// Mitsubishi GX Works2 project: 2023-06-07 #1 생산자동화기능사 13번   PLC: Q03UDV
// 생산자동화기능사

// global labels: Global1
VAR_GLOBAL
  PB1 AT X0 : BOOL;
  PB2 AT X1 : BOOL;
  정지 AT X2 : BOOL;
  공급후진 AT X3 : BOOL;
  공급전진 AT X4 : BOOL;
  가공후진 AT X5 : BOOL;
  가공전진 AT X6 : BOOL;
  송출후진 AT X7 : BOOL;
  송출전진 AT X8 : BOOL;
  배출후진 AT X9 : BOOL;
  배출전진 AT X0A : BOOL;
  매거진 AT X0B : BOOL;
  금속센서 AT X0F : BOOL;
  PB3 AT X10 : BOOL;
  적색 AT Y20 : BOOL;
  황색 AT Y21 : BOOL;
  녹색 AT Y22 : BOOL;
  공급1 AT Y23 : BOOL;
  공급2 AT Y24 : BOOL;
  가공 AT Y25 : BOOL;
  드릴 AT Y26 : BOOL;
  송출 AT Y27 : BOOL;
  배출 AT Y28 : BOOL;
  컨베이어 AT Y29 : BOOL;
END_VAR

PROGRAM 테스트동작
VAR
  prog : INT;
END_VAR
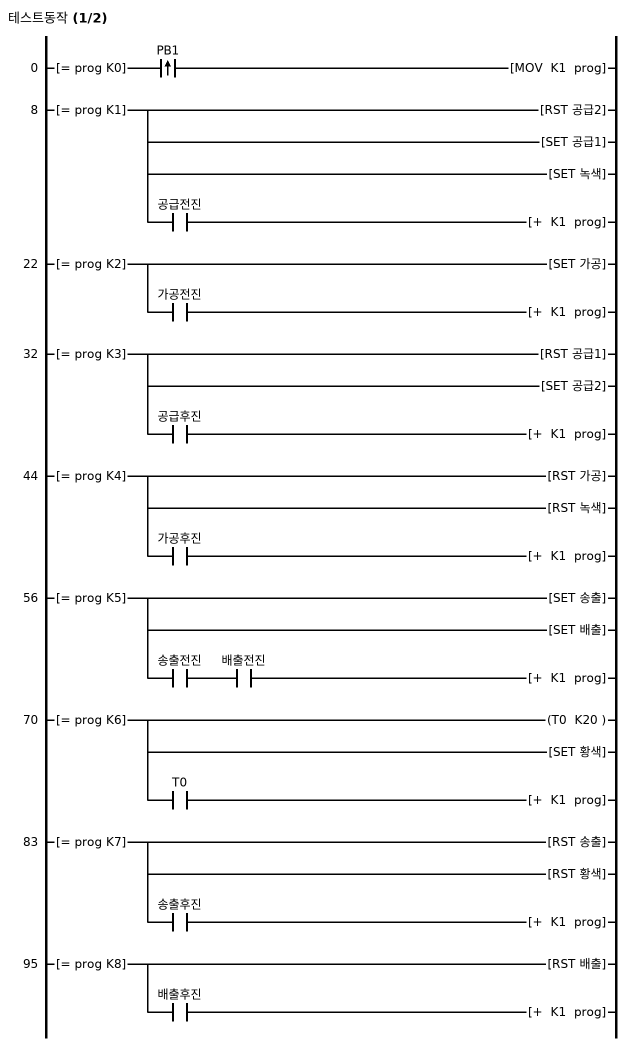
0     LD=     prog K0
      ANDP    PB1
      MOV     K1 prog
8     LD=     prog K1
      RST     공급2
      SET     공급1
      SET     녹색
      AND     공급전진
      +       K1 prog
22    LD=     prog K2
      SET     가공
      AND     가공전진
      +       K1 prog
32    LD=     prog K3
      RST     공급1
      SET     공급2
      AND     공급후진
      +       K1 prog
44    LD=     prog K4
      RST     가공
      RST     녹색
      AND     가공후진
      +       K1 prog
56    LD=     prog K5
      SET     송출
      SET     배출
      AND     송출전진
      AND     배출전진
      +       K1 prog
70    LD=     prog K6
      OUT     T0 K20
      SET     황색
      AND     T0
      +       K1 prog
83    LD=     prog K7
      RST     송출
      RST     황색
      AND     송출후진
      +       K1 prog
95    LD=     prog K8
      RST     배출
      AND     배출후진
      +       K1 prog
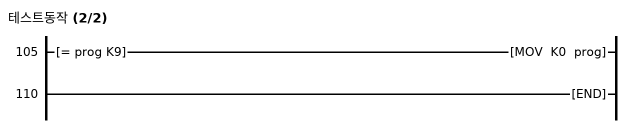
105   LD=     prog K9
      MOV     K0 prog
110   END
END_PROGRAM

PROGRAM 생산자동화기능사
VAR
  prog : INT;
  mode : INT;
END_VAR
VAR CONSTANT
  단속 : INT;
  연속 : INT := 1;
END_VAR
VAR
  metal : INT;
END_VAR
VAR CONSTANT
  금속 : INT := 1;
  비금속 : INT := 2;
END_VAR
VAR
  blink1 : ARRAY [0..3] OF BOOL;
  loop1 : INT;
END_VAR
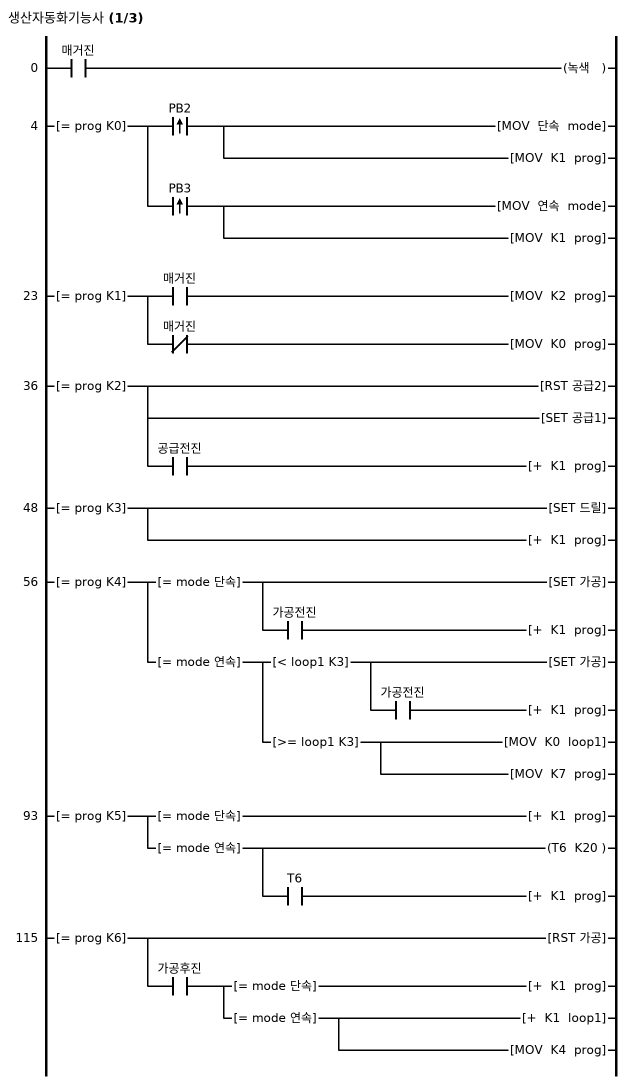
0     LD      매거진
      OUT     녹색
4     LD=     prog K0
      MPS
      ANDP    PB2
      MOV     단속 mode
      MOV     K1 prog
      MPP
      ANDP    PB3
      MOV     연속 mode
      MOV     K1 prog
23    LD=     prog K1
      MPS
      AND     매거진
      MOV     K2 prog
      MPP
      ANI     매거진
      MOV     K0 prog
36    LD=     prog K2
      RST     공급2
      SET     공급1
      AND     공급전진
      +       K1 prog
48    LD=     prog K3
      SET     드릴
      +       K1 prog
56    LD=     prog K4
      MPS
      AND=    mode 단속
      SET     가공
      AND     가공전진
      +       K1 prog
      MPP
      AND=    mode 연속
      MPS
      AND<    loop1 K3
      SET     가공
      AND     가공전진
      +       K1 prog
      MPP
      AND>=   loop1 K3
      MOV     K0 loop1
      MOV     K7 prog
93    LD=     prog K5
      MPS
      AND=    mode 단속
      +       K1 prog
      MPP
      AND=    mode 연속
      OUT     T6 K20
      AND     T6
      +       K1 prog
115   LD=     prog K6
      RST     가공
      AND     가공후진
      MPS
      AND=    mode 단속
      +       K1 prog
      MPP
      AND=    mode 연속
      +       K1 loop1
      MOV     K4 prog
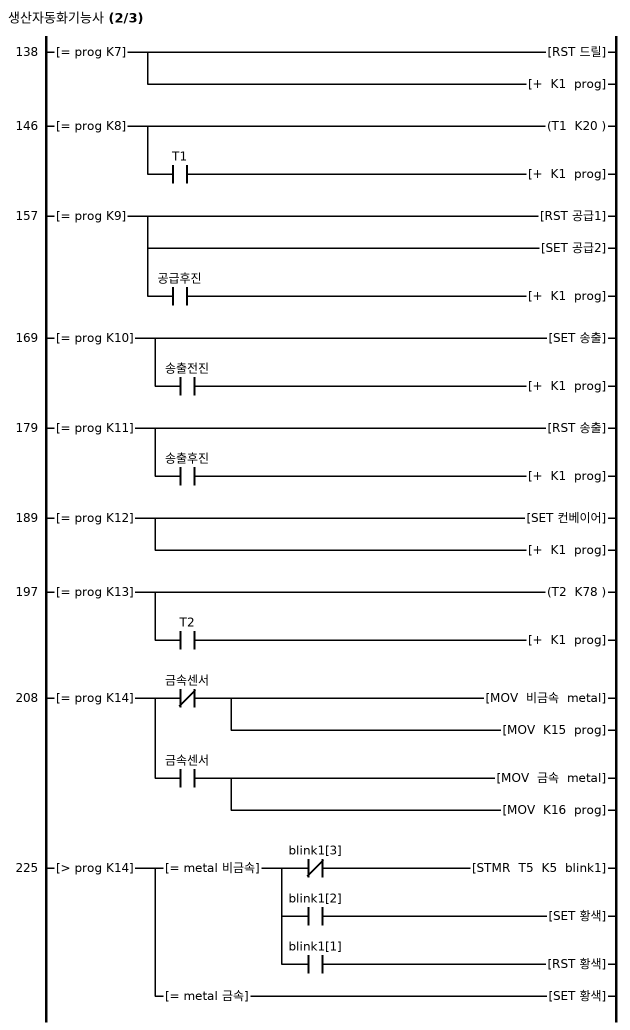
138   LD=     prog K7
      RST     드릴
      +       K1 prog
146   LD=     prog K8
      OUT     T1 K20
      AND     T1
      +       K1 prog
157   LD=     prog K9
      RST     공급1
      SET     공급2
      AND     공급후진
      +       K1 prog
169   LD=     prog K10
      SET     송출
      AND     송출전진
      +       K1 prog
179   LD=     prog K11
      RST     송출
      AND     송출후진
      +       K1 prog
189   LD=     prog K12
      SET     컨베이어
      +       K1 prog
197   LD=     prog K13
      OUT     T2 K78
      AND     T2
      +       K1 prog
208   LD=     prog K14
      MPS
      ANI     금속센서
      MOV     비금속 metal
      MOV     K15 prog
      MPP
      AND     금속센서
      MOV     금속 metal
      MOV     K16 prog
225   LD>     prog K14
      MPS
      AND=    metal 비금속
      MPS
      ANI     blink1[3]
      STMR    T5 K5 blink1
      MRD
      AND     blink1[2]
      SET     황색
      MPP
      AND     blink1[1]
      RST     황색
      MPP
      AND=    metal 금속
      SET     황색
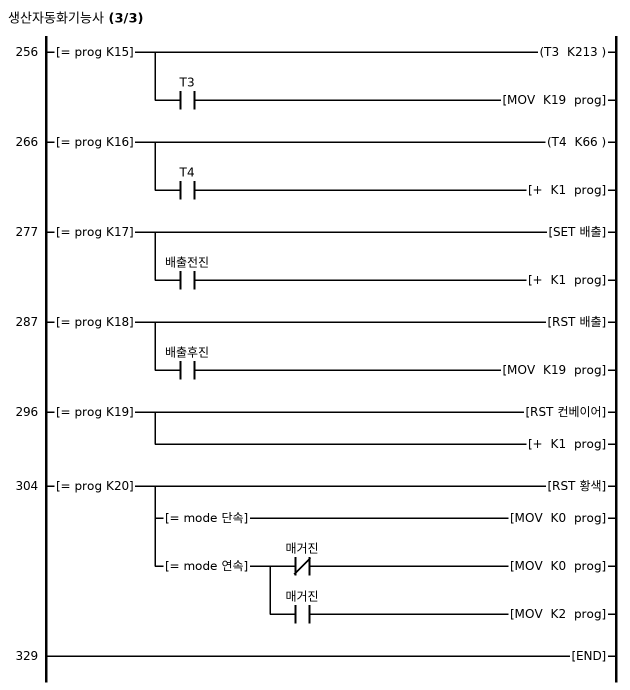
256   LD=     prog K15
      OUT     T3 K213
      AND     T3
      MOV     K19 prog
266   LD=     prog K16
      OUT     T4 K66
      AND     T4
      +       K1 prog
277   LD=     prog K17
      SET     배출
      AND     배출전진
      +       K1 prog
287   LD=     prog K18
      RST     배출
      AND     배출후진
      MOV     K19 prog
296   LD=     prog K19
      RST     컨베이어
      +       K1 prog
304   LD=     prog K20
      RST     황색
      MPS
      AND=    mode 단속
      MOV     K0 prog
      MPP
      AND=    mode 연속
      MPS
      ANI     매거진
      MOV     K0 prog
      MPP
      AND     매거진
      MOV     K2 prog
329   END
END_PROGRAM
